// Mitsubishi GX Works2 project: TCP   PLC: FX3U/FX3UC

PROGRAM MAIN
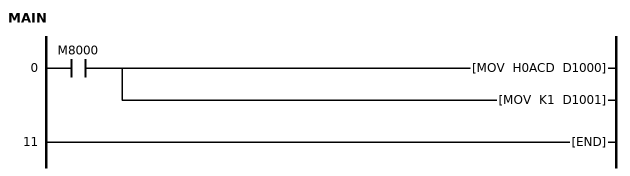
0     LD      M8000
      MOV     H0ACD D1000
      MOV     K1 D1001
11    END
END_PROGRAM

// device comments not shown above
Y020  ; ADP就緒
Y021  ; ADP錯誤
